{attribute 'qualified_only'}
{attribute 'strict'}
TYPE E_SystemControlState :
(
	automatic 	:= 0,
	algorithm	:= 1,
	manual		:= 2
);
END_TYPE

(* stored: Version 1.1.0.1, ProductVersion 3.1.4024.9
   DUT E_SystemControlState: Id {9817809b-cf85-46c9-ae1f-a83f65c089ae} *)
